INTERFACE I_DisSensor

PROPERTY Distance : REAL
GET
END_GET
END_PROPERTY

END_INTERFACE

(* stored: Version 1.1.0.1, ProductVersion 3.1.4024.15
   Itf I_DisSensor: Id {050f86af-adbd-456a-99b1-9194f201a456}
   Property Distance: Id {ed4a445a-f6ea-4bfe-bb8d-fb555743141b}
   Get Get: Id {4d870a83-a994-4a84-87a2-523ad01d0246} *)
